// TIA Portal V18 export
FUNCTION_BLOCK "LGasp_Riordino"   // FB10300, LAD
{ S7_Optimized_Access := 'TRUE' }
VERSION : 0.1
// Da verificare:
// stored: AutoNumber true, IsIECCheckEnabled false, IsRetainMemResEnabled false, MemoryReserve 100, SetENOAutomatically false, UDAEnableTagReadback false
   VAR_INPUT
      i_lista_compilata { ExternalAccessible := 'False'; ExternalVisible := 'False'; ExternalWritable := 'False'} : Bool;   // azzerabuffer riordino e comincia a riordinare
      i_reset : Bool;
      i_svuotamentoDaPC : Bool;   // svuotamento impianto
      i_richTrasfListaPrd { ExternalAccessible := 'False'; ExternalVisible := 'False'; ExternalWritable := 'False'} : Bool;   // richiesta trasferimento lista produzione da PC
      i_mergeAbilitato { ExternalAccessible := 'False'; ExternalVisible := 'False'; ExternalWritable := 'False'} : Bool := false;   // Abilita merge quote
      I_controlloPassoLungo_ON { ExternalAccessible := 'False'; ExternalVisible := 'False'; ExternalWritable := 'False'} : Bool;   // abilita controllo passo lungo
      i_lunghezzaBanco { ExternalAccessible := 'False'; ExternalVisible := 'False'; ExternalWritable := 'False'} : LReal;
      i_quotaPrimaPunzonata { ExternalVisible := 'False'; ExternalWritable := 'False'} : LReal;
      i_correttore { ExternalVisible := 'False'; ExternalWritable := 'False'} : LReal := 1.0;
      i_passoLungoMax { ExternalVisible := 'False'; ExternalWritable := 'False'} : LReal;   // passo massimo (utilizzato per alimentatori a rulli)
   END_VAR
   VAR_OUTPUT
      o_quote_OK { ExternalAccessible := 'False'; ExternalVisible := 'False'; ExternalWritable := 'False'} : Bool;
      o_lim_max_quote { ExternalAccessible := 'False'; ExternalVisible := 'False'; ExternalWritable := 'False'} : Bool;   // raggiunto limite quote su riordino (incrementare costante "NumQuotePunzonatura" )
      o_OkTrasfListaPrd : Bool;
      o_AlmPreFineQuote : Bool;
      o_AlmFineQuote : Bool;
      o_QuotaAssoluta : "LGasp_typeBufferQuote";   // Quota assoluta
      o_QuotaAssoluta_Correttore : "LGasp_typeBufferQuote";   // Quota assoluta
      o_QuotaRelativa : "LGasp_typeBufferQuote";   // Quota relativa
      o_QuotaRelativa_Correttore : "LGasp_typeBufferQuote";   // Quota relativa con correttore
   END_VAR
   VAR_IN_OUT
      io_PunzonataEseguita { ExternalAccessible := 'False'; ExternalVisible := 'False'; ExternalWritable := 'False'} : Bool;   // cancella quota in lavoro
      io_cancella_pezzi : Bool;   // cmdbool00[8]
      io_lista_profila_nuovo_elemento : Bool;
      io_cancellazioneTotale : Bool;   // cmdbool00[11]
      io_blocca_lista_fine_prod : Bool;
      io_rich_nuovo_trasferimento : Bool;   // richiesta nuovo trasferimento all'avvio
      io_PassoInfinito : "LGasp_typeQuota";
      io_ListaProduzionePC : Array[1.."NumRigheProduzione"] of "LGasp_typeRigaProdfromPC";
      io_myprodfromPC : Array[1.."NumRigheProduzione"] of "LGasp_typeRigaProdfromPC";
      io_myprodfromPCupdate : Array[1.."NumRigheProduzione"] of DInt;
      io_myprodfromPLC : Array[1.."NumRigheProduzione"] of "LGasp_typeRigaProdfromPLC";
      io_StoricoQuotePunzonatura : Array[1.."NumQuotePunzonaturaStorico"] of "LGasp_typeBufferQuote";
      io_QuotePunzonatura : Array[1.."NumQuotePunzonatura"] of "LGasp_typeBufferQuote";
      io_StoricoRigheProdEliminate : Array[1.."NumRigheProduzione"] of "LGasp_typeRigheEliminate";
      io_pezzo_per_Lista_profila : "LGasp_typePzoListaProfila";
   END_VAR
   VAR RETAIN
      s_DM { ExternalAccessible := 'False'; ExternalVisible := 'False'; ExternalWritable := 'False'} : Struct
         OffsetPrimaPunzonata { ExternalAccessible := 'False'; ExternalVisible := 'False'; ExternalWritable := 'False'} : LReal := 0.0;   // Quota prima punzonata dopo ricompilazione
      END_STRUCT;
   END_VAR
   VAR
      s_RiordinoBufferQuote_QuickSort { ExternalAccessible := 'False'; ExternalVisible := 'False'; ExternalWritable := 'False'} : "LGasp_RiordinoBufferQuote_QuickSort";
      "s_Aggiorna&Riordina" { ExternalAccessible := 'False'; ExternalVisible := 'False'; ExternalWritable := 'False'} : Bool;   // aggiorna quote e riordina
   END_VAR
   VAR RETAIN
      s_start_riordino { ExternalAccessible := 'False'; ExternalVisible := 'False'; ExternalWritable := 'False'} : Bool;
      s_sort_riordino_OK { ExternalAccessible := 'False'; ExternalVisible := 'False'; ExternalWritable := 'False'} : Bool;
      s_lista_compilata_old { ExternalAccessible := 'False'; ExternalVisible := 'False'; ExternalWritable := 'False'} : Bool;
      s_inserire_pezzi_in_lista { ExternalAccessible := 'False'; ExternalVisible := 'False'; ExternalWritable := 'False'} : Bool;   // inserire pezzi in lista produzione
   END_VAR
   VAR
      s_firstscan_done { ExternalAccessible := 'False'; ExternalVisible := 'False'; ExternalWritable := 'False'} : Bool;
      s_ListaProduzione_ID_old { ExternalAccessible := 'False'; ExternalVisible := 'False'; ExternalWritable := 'False'} : Array[1.."NumRigheProduzione"] of DInt;
      s_index_0 { ExternalAccessible := 'False'; ExternalVisible := 'False'; ExternalWritable := 'False'} : DInt;
      s_index_1 { ExternalAccessible := 'False'; ExternalVisible := 'False'; ExternalWritable := 'False'} : DInt;
      s_index_2 { ExternalAccessible := 'False'; ExternalVisible := 'False'; ExternalWritable := 'False'} : DInt;
      s_index_3 { ExternalAccessible := 'False'; ExternalVisible := 'False'; ExternalWritable := 'False'} : DInt;
      s_index_4 { ExternalAccessible := 'False'; ExternalVisible := 'False'; ExternalWritable := 'False'} : DInt;
      s_index_5 { ExternalAccessible := 'False'; ExternalVisible := 'False'; ExternalWritable := 'False'} : DInt;
      s_index_6 { ExternalAccessible := 'False'; ExternalVisible := 'False'; ExternalWritable := 'False'} : DInt;
      s_index_7 { ExternalAccessible := 'False'; ExternalVisible := 'False'; ExternalWritable := 'False'} : DInt;
   END_VAR
   VAR RETAIN
      s_RigaProduzione_in_lavoro { ExternalAccessible := 'False'; ExternalVisible := 'False'; ExternalWritable := 'False'} : DInt;   // Indice riga di produzione in lavoro
      s_PrimaQuotaLibera { ExternalAccessible := 'False'; ExternalVisible := 'False'; ExternalWritable := 'False'} : DInt;   // Indice della prima quota NULL nella DB di riordino Quote
      s_quote_inserite { ExternalAccessible := 'False'; ExternalVisible := 'False'; ExternalWritable := 'False'} : DInt;
      s_lunghezza { ExternalAccessible := 'False'; ExternalVisible := 'False'; ExternalWritable := 'False'} : LReal;   // appoggio lunghezza pezzo i inserimento
      s_lunghezza_tot_inserita_banco { ExternalAccessible := 'False'; ExternalVisible := 'False'; ExternalWritable := 'False'} : LReal;   // lunghezza banco per inserimento pezzi
      s_tot_materiale_inserito_dopo_compilazione { ExternalAccessible := 'False'; ExternalVisible := 'False'; ExternalWritable := 'False'} : LReal;   // totale materiale inserito dopo compilazione
   END_VAR
   VAR
      s_lunghezza_banco { ExternalAccessible := 'False'; ExternalVisible := 'False'; ExternalWritable := 'False'} : LReal;
      s_QuotaNULL { ExternalAccessible := 'False'; ExternalVisible := 'False'; ExternalWritable := 'False'} : "LGasp_typeQuota";   // tipo dato NULL
      s_BufferQuotaNULL { ExternalAccessible := 'False'; ExternalVisible := 'False'; ExternalWritable := 'False'} : "LGasp_typeBufferQuote";   // tipo dato NULL
      s_RigaProduzioneNULL { ExternalAccessible := 'False'; ExternalVisible := 'False'; ExternalWritable := 'False'} : "LGasp_typeRigaProdfromPC";   // tipo dato NULL
      s_mem_trasf_lista_da_PC { ExternalAccessible := 'False'; ExternalVisible := 'False'; ExternalWritable := 'False'} : Bool;
   END_VAR
   VAR RETAIN
      s_ID_righe_produzione { ExternalAccessible := 'False'; ExternalVisible := 'False'; ExternalWritable := 'False'} : Array[1.."NumRigheProduzione"] of DInt;
      s_quotaTestaInserita { ExternalAccessible := 'False'; ExternalVisible := 'False'; ExternalWritable := 'False'} : Bool;
      s_mem_quota { ExternalAccessible := 'False'; ExternalVisible := 'False'; ExternalWritable := 'False'} : LReal;
      s_appQuota { ExternalAccessible := 'False'; ExternalVisible := 'False'; ExternalWritable := 'False'} : LReal;
      s_count { ExternalAccessible := 'False'; ExternalVisible := 'False'; ExternalWritable := 'False'} : DInt;
      s_num_pzi_banco { ExternalAccessible := 'False'; ExternalVisible := 'False'; ExternalWritable := 'False'} : Int;
   END_VAR
   VAR
      s_FPPreFine { ExternalAccessible := 'False'; ExternalVisible := 'False'; ExternalWritable := 'False'} : Bool;
      s_ResetPassoInfinito { ExternalAccessible := 'False'; ExternalVisible := 'False'; ExternalWritable := 'False'} : Bool;
      s_primoTrasferimentoEseguito { ExternalAccessible := 'False'; ExternalVisible := 'False'; ExternalWritable := 'False'} : Bool;
      s_passoLungoON : Bool;
   END_VAR
   VAR_TEMP
      t_passoLungoMax : LReal;
   END_VAR
   VAR_TEMP   // added for the SCL form of the ladder/FBD networks
      _w1 : Bool;
   END_VAR
BEGIN

REGION Network 1 (SCL): Descrizione
   //================================================================================
   // Gasparini Spa
   //--------------------------------------------------------------------------------
   // Libreria: LGaspQset_Riordino
   // Funzionalità: Funzione globale per gestione riordino quote
   // Commessa in cui è stata testata: YYXXNNNNN
   // Programmatore di riferimento per test: XXXXXX
   //--------------------------------------------------------------------------------
   // Change log table:
   // Versione Data        Autore          Modifiche
   // 01.00.03 02.07.2020  P.Toaldo        Aggiornamento dopo test quote con PC
   // 01.00.04 22/03/2021  Lcg             Banco di punzonatura per calcoli quote deve essere il doppio di quello reale
   // 01.00.05 08/04/2021  Lcg             Inserito un pulsante da PC che esegue la cancellazione totale
   // 01.00.06 27/05/2021  P.Toaldo        Correzione aggiornamento quota dopo set "io_PunzonataEseguita". Micron 305
   // 01.00.06 27/05/2021  Lcg             Correzione uscita "Sort" blocco riordino che non era ritentiva  Micron 305
   // 01.00.07 03/06/2021  Lcg             Correzione errore prefine lista e aggiunto blocco lista di produzione a fine pezzi
   // 01.00.08 10/06/2021  Lcg             Reset passo infinito con cancellazione lista
   // 01.00.09 28/06/2021  Lcg             Corretto errore cancellazione passo infinito con nuova compilazione
   // 01.00.10 06/07/2021  Lcg             Corretto errore nuovo trasferimento all'avvio del PC seg 18
   // 01.00.11 28/01/2022  Lcg             Aggiunto il reset dell'area di memoria passo infinito con primo trasferimento e lista non compilata
   // 01.00.12 02/03/2022  Lcg/A.Donà      Aggiunto il numero del pezzo a cui fa riferimento la quota. In state aggiunto se la quota è una quota di sincronismo.
   //                                      Aggiunto nome articolo nella struttura per passaggio a lista profila e ad eventuale tracking (210100012)
   // 01.00.13 10/10/2022  Lcg             Passaggio nuovi dati option.DINT, options.Lreal, options.Str in lista profila
   // 01.00.14 24/01/2023  Lcg             Aggiunto "i_quotaPrimaPunzonata" alla prima quota se era un passo infinito perchè non veniva sommata
   // 01.00.15 14/03/2023  Lcg             Corretto errore che all'avvio azzerava i pezzi fatti dopo uno snapshot di L1_prd (22010003)
   // 01.00.16 17/03/2023  Lcg             Eliminata la funzionalità lunghezza pezzi non multipla del passo alimentatore usata solo su Micron 303 perchè creava confusione con lenght e nominal lenght 
   //                                      in quanto lenght comprende lo sfrido e nominal lenght è senza sfrido. Questo causava un errore nella visualizzazione del numero pezzo della lista profila.
   //                                      Corretto errore "Allarme fine pezzi" all'accensione, si attende il primo trasferimento. 
   // 01.00.17 20/04/2023  Lcg             Aggiunta gestione passo lungo, si può abilitare una funzione che in caso di quota maggiore di i_passoLungoMax la quota viene ridotta
   //                                      in sottopassi di grandezza massima i_passoLungoMax (SIPPA 220100034). Passo lungo e passo infinito non possono coesistere.
   // 01.00.18 09/05/2023  Lcg             Modificato blocco inserimento righe PC dopo preavviso fine lista perchè se veniva premuto reset prima di inserire la riga non era più possibile
   //                                      eseguire l'inserimento (dierre 210100104)
   // 
   //-------------------------------------------------------------------------------
   //================================================================================
END_REGION

REGION Network 2 (SCL): Lunghezza banco di punzonatura + quota primapunzonata
   // la lunghezza del banco di punzonatura sul nuovo riordino quote deve essere uguale alla lunghezza reale del banco per 2 altrimenti possono capitare casi per cui l'inserimento delle nuove quote è tardivo
   //lunghezza banco
   #s_lunghezza_banco := #i_lunghezzaBanco * 2.0;

   //quota prima punz
   #s_DM.OffsetPrimaPunzonata := #i_quotaPrimaPunzonata;

   //valore quota/passo massimo
   #t_passoLungoMax := #i_passoLungoMax;
END_REGION

REGION Network 3 (SCL): Appoggio Produzione dal PC sulla produzione del PLC


   IF #i_richTrasfListaPrd THEN
       #s_mem_trasf_lista_da_PC := TRUE;
   END_IF;

   IF NOT #i_richTrasfListaPrd AND #s_mem_trasf_lista_da_PC THEN
       #s_mem_trasf_lista_da_PC := FALSE;
       #io_myprodfromPC :=  #io_ListaProduzionePC;
   END_IF;
END_REGION

REGION Network 4 (SCL): Su fronte compilazione lista -> cancello tutto il DB riordino quote e lancio riordino
   IF #i_lista_compilata AND (NOT #s_lista_compilata_old) AND NOT #i_richTrasfListaPrd THEN

       FOR #s_index_1 := 1 TO "NumQuotePunzonatura" DO // Statement section IF
           #io_QuotePunzonatura[#s_index_1] := #s_BufferQuotaNULL;
       END_FOR;

       // cancella storico
       FOR #s_index_1 := 1 TO "NumQuotePunzonaturaStorico" DO // Statement section IF
           #io_StoricoQuotePunzonatura[#s_index_1] := #s_BufferQuotaNULL;
       END_FOR;

       // Aggiorno il numero di pezzi inseriti nel riordino quote = pezzi fatti
       FOR #s_index_1 := 1 TO "NumRigheProduzione" DO
           #io_myprodfromPLC[#s_index_1].pzinseritinelriordinoquote := #io_myprodfromPLC[#s_index_1].pzfatti;
       END_FOR;
       #s_tot_materiale_inserito_dopo_compilazione := #s_DM.OffsetPrimaPunzonata;
       #s_lunghezza_tot_inserita_banco := 0.0;
       #s_quotaTestaInserita := False;
       #s_passoLungoON := false;
       #s_num_pzi_banco := 0;

       #"s_Aggiorna&Riordina" := true;
   END_IF;

   IF #i_lista_compilata = false AND #s_lista_compilata_old = true THEN

       FOR #s_index_1 := 1 TO "NumQuotePunzonatura" DO // Statement section IF
           #io_QuotePunzonatura[#s_index_1] := #s_BufferQuotaNULL;
       END_FOR;

       // Aggiorno il numero di pezzi inseriti nel riordino quote = pezzi fatti
       FOR #s_index_1 := 1 TO "NumRigheProduzione" DO
           #io_myprodfromPLC[#s_index_1].pzinseritinelriordinoquote := #io_myprodfromPLC[#s_index_1].pzfatti;
       END_FOR;

       #s_tot_materiale_inserito_dopo_compilazione := #s_DM.OffsetPrimaPunzonata;
       #s_lunghezza_tot_inserita_banco := 0.0;
       #s_quotaTestaInserita := False;
       #s_passoLungoON := false;
       #s_num_pzi_banco := 0;

   END_IF;

   #s_lista_compilata_old := #i_lista_compilata;
END_REGION

REGION Network 5 (SCL): Cancellazione totale da pulsante in pagina di produzione che esegue la cancellazione totale
       IF #io_cancellazioneTotale THEN

           //cancella quote punzonatura
           FOR #s_index_1 := 1 TO "NumQuotePunzonatura" DO // Statement section IF
               #io_QuotePunzonatura[#s_index_1] := #s_BufferQuotaNULL;
           END_FOR;

           //cancello tutto
           FOR #s_index_1 := 1 TO "NumRigheProduzione" DO
               #io_myprodfromPLC[#s_index_1].pzinseritinelriordinoquote := 0;
               #io_myprodfromPLC[#s_index_1].pzfatti := 0;

               #io_myprodfromPC[#s_index_1].ID := 0;
               #io_myprodfromPC[#s_index_1].piecestodo := 0;
               #io_myprodfromPC[#s_index_1].tipoarticolo := 0;

           END_FOR;

           #io_cancellazioneTotale := false;

       END_IF;
END_REGION

REGION Network 6 (SCL): Cancellazione aree passo infinito con primo trasferimento e lista non compilata in quanto il PC non le cancella
           //Nessun trasferimento in corso
           IF NOT #i_richTrasfListaPrd THEN
               #s_ResetPassoInfinito := false;
           END_IF;

           //con fronte trasferimento e lista non compilata azzero l'area del passo infinito
           IF NOT #i_lista_compilata AND #i_richTrasfListaPrd AND NOT #s_ResetPassoInfinito THEN

               #s_ResetPassoInfinito := true;

               //reset passo infinito 
               #io_PassoInfinito.quotax := -1;
               #io_PassoInfinito.quotay := -1;

               //reset dei punzoni del passo infinito
               FOR #s_index_1 := 1 TO 16 DO
                   #io_PassoInfinito.mouldea[#s_index_1] := false;
                   #io_PassoInfinito.mouldeb[#s_index_1] := false;
                   #io_PassoInfinito.mouldec[#s_index_1] := false;
                   #io_PassoInfinito.moulded[#s_index_1] := false;
               END_FOR;

               #io_PassoInfinito.infinitystep := false;

           END_IF;
END_REGION

REGION Network 7 (SCL): Riga di produzione in lavoro
   FOR #s_index_1 := 1 TO "NumRigheProduzione" DO
       IF #io_myprodfromPLC[#s_index_1].pzfatti < #io_myprodfromPC[#s_index_1].piecestodo THEN
           #s_RigaProduzione_in_lavoro := #s_index_1;
           EXIT;
       END_IF;
   END_FOR;
END_REGION

REGION Network 8 (SCL): Prima quota libera nel DB di riordino quote
   FOR #s_index_1 := 1 TO "NumQuotePunzonatura" DO
       IF NOT(#io_QuotePunzonatura[#s_index_1].quota.state.quotavalida) THEN
           #s_PrimaQuotaLibera := #s_index_1;
           EXIT;
       END_IF;
   END_FOR;
END_REGION

REGION Network 9: Reset allarme limite massimo quote inserite con togli compilazione
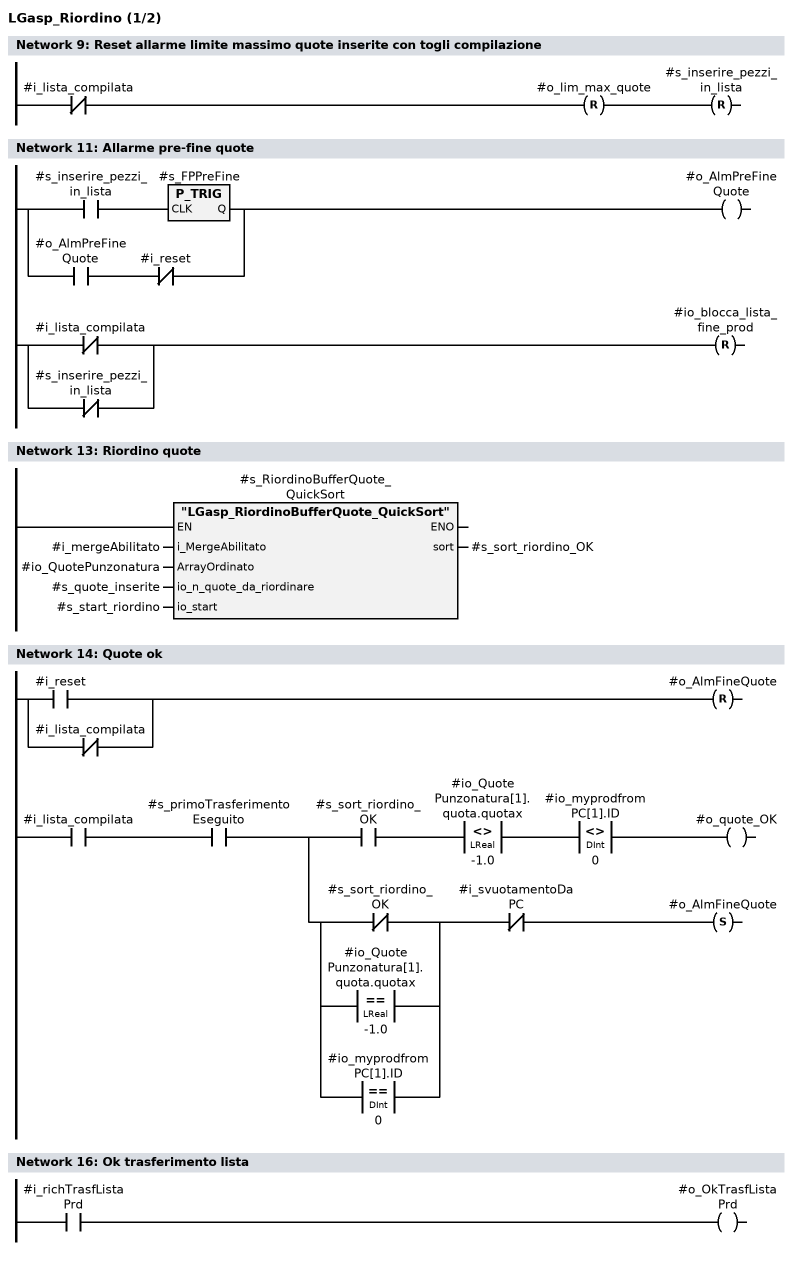
   RUNG wire#powerrail
      I_Contact( #i_lista_compilata )
      R_Coil( #o_lim_max_quote )
      R_Coil( #s_inserire_pezzi_in_lista )
   END_RUNG
   // the same network as SCL:
   IF NOT #i_lista_compilata THEN
       #o_lim_max_quote := FALSE;
       #s_inserire_pezzi_in_lista := FALSE;
   END_IF;
END_REGION

REGION Network 10 (SCL): Lista quote con le quote con articoli fino a riempire la lunghezza del banco di punzonatura
   // rilancio controllo per verifica pre-fine quote
   IF #i_reset AND #o_AlmPreFineQuote THEN
       #"s_Aggiorna&Riordina" := TRUE;
   END_IF;


   IF #"s_Aggiorna&Riordina" AND #s_primoTrasferimentoEseguito THEN
       #io_PunzonataEseguita := false;
       #s_inserire_pezzi_in_lista := false;
       #s_quote_inserite := #s_PrimaQuotaLibera - 1;



       // Se presente passo infinito inserisco la prima quota
       IF #s_quote_inserite = 0 AND #io_PassoInfinito.infinitystep THEN

           // INSERISCO QUOTA SU RIORDINO
           #s_quote_inserite := #s_quote_inserite + 1;
           #io_QuotePunzonatura[#s_quote_inserite].quota := #io_PassoInfinito;
           //24.01.2023 lcg
           //aggiungo prima quota al primo passo infinito
           #io_QuotePunzonatura[#s_quote_inserite].quota.quotax := #io_QuotePunzonatura[#s_quote_inserite].quota.quotax + #i_quotaPrimaPunzonata;

       END_IF;

       //verifico se la prima quota supera il passo massimo 
       IF #s_quote_inserite = 0 AND #I_controlloPassoLungo_ON AND NOT #io_PassoInfinito.infinitystep AND NOT #s_passoLungoON THEN

           #s_appQuota := #io_myprodfromPC[1].article.prepunchingquota[1].quotax + #i_quotaPrimaPunzonata;

           IF #s_appQuota > #i_passoLungoMax THEN

               // INSERISCO QUOTA SU RIORDINO

               #s_quote_inserite := #s_quote_inserite + 1;
               //cancello tutti i cassetti
               #io_QuotePunzonatura[1].quota := #s_QuotaNULL;
               #io_QuotePunzonatura[#s_quote_inserite].quota.quotax := #i_passoLungoMax;
               #s_passoLungoON := true;

           END_IF;
       END_IF;

       // Inserisco le quote degli articoli fino al riempimento del banco di punzonatura
       FOR #s_index_1 := 1 TO "NumRigheProduzione" DO
           IF #io_myprodfromPLC[#s_index_1].pzinseritinelriordinoquote < #io_myprodfromPC[#s_index_1].piecestodo THEN
               FOR #s_index_2 := #io_myprodfromPLC[#s_index_1].pzinseritinelriordinoquote + 1 TO #io_myprodfromPC[#s_index_1].piecestodo DO
                   IF #s_lunghezza_tot_inserita_banco < #s_lunghezza_banco OR #s_num_pzi_banco < 2 THEN
                       // Inserisco tutte le punzonate dell'articolo in riga di produzione
                       FOR #s_index_3 := 1 TO "NumPunzonateArticolo" DO

                           // Controllo che la quota dell'articolo sia valida
                           IF #io_myprodfromPC[#s_index_1].article.prepunchingquota[#s_index_3].state.quotavalida AND NOT (#o_lim_max_quote)  THEN

                               //24.01.2023 Lcg: Tolta l'istruzione che non metteva nel riordino le quote di testa dopo la prima (Dierre 104)
                               //IF (NOT #s_quotaTestaInserita OR NOT #io_myprodfromPC[#s_index_1].article.prepunchingquota[#s_index_3].state.quotatagliotesta) THEN

                                   IF #io_myprodfromPC[#s_index_1].article.prepunchingquota[#s_index_3].state.quotatagliotesta THEN
                                       #s_quotaTestaInserita := TRUE;
                                   END_IF;

                                   // incrementa quote inserite
                                   #s_quote_inserite := #s_quote_inserite + 1;

                                   // Aggiorno articolo, general , quota e testo stampa

                                   #io_QuotePunzonatura[#s_quote_inserite].general := #io_myprodfromPC[#s_index_1].article.general;
                                   #io_QuotePunzonatura[#s_quote_inserite].quota := #io_myprodfromPC[#s_index_1].article.prepunchingquota[#s_index_3];
                                   #io_QuotePunzonatura[#s_quote_inserite].general.print := #io_myprodfromPC[#s_index_1].article.general.print;
                                   #io_QuotePunzonatura[#s_quote_inserite].ID := #io_myprodfromPC[#s_index_1].ID;
                                   //numero del pezzo a cui fa riferimento la quota
                                   #io_QuotePunzonatura[#s_quote_inserite].n_piece := #s_index_2;

                                   // alla quota X aggiungo l'offset di partenza
                                   #io_QuotePunzonatura[#s_quote_inserite].quota.quotax := (#io_QuotePunzonatura[#s_quote_inserite].quota.quotax) + #s_tot_materiale_inserito_dopo_compilazione;



                                   // memorizzo lunghezza pezzo dell'ultima quota
                                   IF #io_QuotePunzonatura[#s_quote_inserite].quota.state.ultimaquotapezzo THEN
                                       #s_lunghezza := #io_QuotePunzonatura[#s_quote_inserite].general.lenght;
                                       EXIT;
                                   END_IF;

                                   // verifica limite quote nel riordino raggiunte
                                   IF #s_quote_inserite >= "NumQuotePunzonatura" THEN
                                       #o_lim_max_quote := TRUE;
                                   END_IF;
                               //END_IF;
                           ELSE
                               EXIT;
                           END_IF;
                       END_FOR;

                       // Aggiungo un pezzo ai pezzi presi in carico dal riordino quote per la riga di produzione in lavoro
                       #io_myprodfromPLC[#s_index_1].pzinseritinelriordinoquote := #io_myprodfromPLC[#s_index_1].pzinseritinelriordinoquote + 1;

                       // aggiorno totale materiale inserito in banco di punzonatura
                       #s_lunghezza_tot_inserita_banco := #s_lunghezza_tot_inserita_banco + #s_lunghezza ;
                       #s_num_pzi_banco := #s_num_pzi_banco+1;

                       // aggiorno totale materiale inserito da dopo compilazione
                       #s_tot_materiale_inserito_dopo_compilazione := #s_tot_materiale_inserito_dopo_compilazione + #s_lunghezza;

                   END_IF;
               END_FOR;
           END_IF;
       END_FOR;

       // verifica fine pezzi
       IF #s_lunghezza_tot_inserita_banco < #s_lunghezza_banco OR #s_num_pzi_banco<2 THEN
           #s_inserire_pezzi_in_lista := true;
       END_IF;



       // comando riordino quote
       #"s_Aggiorna&Riordina" := FALSE;
       #s_start_riordino := true;
   END_IF;
END_REGION

REGION Network 11: Allarme pre-fine quote
   RUNG wire#powerrail
      Contact( #s_inserire_pezzi_in_lista )
      P_Trig( #s_FPPreFine )
      wire#w1
      Coil( #o_AlmPreFineQuote )
   END_RUNG
   RUNG wire#powerrail
      Contact( #o_AlmPreFineQuote )
      I_Contact( #i_reset )
   END_RUNG wire#w1
   RUNG wire#powerrail
      I_Contact( #i_lista_compilata )
      wire#w2
      R_Coil( #io_blocca_lista_fine_prod )
   END_RUNG
   RUNG wire#powerrail
      I_Contact( #s_inserire_pezzi_in_lista )
   END_RUNG wire#w2
   // the same network as SCL:
   #_w1 := #s_inserire_pezzi_in_lista AND NOT #s_FPPreFine;   // rising edge
   #s_FPPreFine := #s_inserire_pezzi_in_lista;
   #o_AlmPreFineQuote := #_w1 OR (#o_AlmPreFineQuote AND NOT #i_reset);
   IF NOT #i_lista_compilata OR NOT #s_inserire_pezzi_in_lista THEN
       #io_blocca_lista_fine_prod := FALSE;
   END_IF;
END_REGION

REGION Network 12 (SCL): Quota eseguita + inserimento nuova quota + riordino
   // comando quota eseguita ->
   // 1 - popolare il DB StoricoQuotePunzonatura con la quota appena cancellata
   // 2 - verificare se è l'ultima quota del pezzo
   // 3 - cancellare prima quota della lista punzonatura

   IF #io_PunzonataEseguita THEN
       #s_count := #s_count + 1;

       // ****************************************
       // aggiornamento DB StoricoQuotePunzonatura 
       // ****************************************

       // Shifto array di un posto per liberare il primo record dell'array
       // NB: record [1] è il più recente
       FOR #s_index_1 := "NumQuotePunzonaturaStorico" TO 2 BY -1 DO
           #io_StoricoQuotePunzonatura[#s_index_1] := #io_StoricoQuotePunzonatura[#s_index_1 - 1];
       END_FOR;

       // Scrivo il primo record dell'array = quota da cancellare
       #io_StoricoQuotePunzonatura[1] := #io_QuotePunzonatura[1];

       // verifico se è l'ultima quota del pezzo
       IF #io_QuotePunzonatura[1].quota.state.ultimaquotapezzo THEN

           // aggiona dati per lista profila
           #io_pezzo_per_Lista_profila.ID := #io_QuotePunzonatura[1].ID;

           //gestione lista profila con articolo a passo e non a passo
           //articolo a passo dello stampo
           //modalità usata in micron 303 dove la lunghezza del pezzo era diversa dal passo fisso dell'alimentatore
           //IF (#io_QuotePunzonatura[1].general.lenght = #io_QuotePunzonatura[1].general.nominal_lenght) OR #io_QuotePunzonatura[1].general.nominal_lenght = -1.0 THEN
           //    #io_pezzo_per_Lista_profila.lenght := #io_QuotePunzonatura[1].general.lenght;
           #io_pezzo_per_Lista_profila.NumeroPezzo := #io_myprodfromPLC[1].pzfatti + 1;
           //ELSE
           //articolo non a passo dello stampo
           #io_pezzo_per_Lista_profila.lenght := #io_QuotePunzonatura[1].general.nominal_lenght;
           //   #io_pezzo_per_Lista_profila.NumeroPezzo := #io_myprodfromPLC[1].pzfattinopasso + 1;
           //END_IF;

           #io_pezzo_per_Lista_profila.cutoffset := #io_QuotePunzonatura[1].general.cutoffset;
           #io_pezzo_per_Lista_profila.options := #io_QuotePunzonatura[1].general.options;
           #io_pezzo_per_Lista_profila.options_dint := #io_myprodfromPC[#s_RigaProduzione_in_lavoro].article.general.options_dint;
           #io_pezzo_per_Lista_profila.options_lreal := #io_myprodfromPC[#s_RigaProduzione_in_lavoro].article.general.options_lreal;
           #io_pezzo_per_Lista_profila.options_str := #io_myprodfromPC[#s_RigaProduzione_in_lavoro].article.general.options_str;
           #io_lista_profila_nuovo_elemento := true;

           // incremento pezzi fatti
           #io_myprodfromPLC[#s_RigaProduzione_in_lavoro].pzfatti := #io_myprodfromPLC[#s_RigaProduzione_in_lavoro].pzfatti + 1;
           // aggiorna lunghezza totale inserita su banco punzonatura
           #s_lunghezza_tot_inserita_banco := #s_lunghezza_tot_inserita_banco - #io_QuotePunzonatura[1].general.lenght;
           #s_num_pzi_banco := #s_num_pzi_banco - 1;
       END_IF;

       // se quota passo infinito riaggiungo la quota altrimenti la elimino
       IF NOT #I_controlloPassoLungo_ON THEN

           // se quota passo infinito riaggiungo la quota altrimenti la elimino
           IF #io_QuotePunzonatura[1].quota.infinitystep THEN

               #s_mem_quota := #io_QuotePunzonatura[1].quota.quotax;
               #io_QuotePunzonatura[1].quota := #io_PassoInfinito;
               #io_QuotePunzonatura[1].quota.quotax := #s_mem_quota + #io_PassoInfinito.quotax;

           ELSE
               FOR #s_index_6 := 1 TO "NumQuotePunzonatura" - 1 DO
                   #io_QuotePunzonatura[#s_index_6] := #io_QuotePunzonatura[#s_index_6 + 1];
               END_FOR;
               #io_QuotePunzonatura[NumQuotePunzonatura] := #s_BufferQuotaNULL;
           END_IF;

       ELSE

           //entro qui se ho il controllo passo lungo
           IF ((#io_QuotePunzonatura[2].quota.quotax - #io_QuotePunzonatura[1].quota.quotax) > #i_passoLungoMax) AND #io_QuotePunzonatura[2].quota.quotax > 0.0 THEN

               //appoggio quota
               #s_mem_quota := #io_QuotePunzonatura[1].quota.quotax;
               //cancello tutti i cassetti
               #io_QuotePunzonatura[1].quota := #s_QuotaNULL;
               #io_QuotePunzonatura[1].quota.quotax := #s_mem_quota + #i_passoLungoMax;

           ELSE
               FOR #s_index_6 := 1 TO "NumQuotePunzonatura" - 1 DO
                   #io_QuotePunzonatura[#s_index_6] := #io_QuotePunzonatura[#s_index_6 + 1];
               END_FOR;
               #io_QuotePunzonatura[NumQuotePunzonatura] := #s_BufferQuotaNULL;
           END_IF;

       END_IF;

       // comando aggiornamento quote + riordino
       #"s_Aggiorna&Riordina" := true;

       //blocco inserimento righe dopo ripartenza e prefine quote attivo
       IF #s_inserire_pezzi_in_lista AND NOT #o_AlmPreFineQuote THEN
           #io_blocca_lista_fine_prod := true;
       END_IF;

   END_IF;
END_REGION

REGION Network 13: Riordino quote
   RUNG wire#powerrail
      #s_RiordinoBufferQuote_QuickSort(i_MergeAbilitato := #i_mergeAbilitato, ArrayOrdinato := #io_QuotePunzonatura, io_n_quote_da_riordinare := #s_quote_inserite, io_start := #s_start_riordino, sort => #s_sort_riordino_OK)
   END_RUNG
   // the same network as SCL:
   #s_RiordinoBufferQuote_QuickSort(i_MergeAbilitato := #i_mergeAbilitato,   // "LGasp_RiordinoBufferQuote_QuickSort"
                           ArrayOrdinato := #io_QuotePunzonatura,
                           io_n_quote_da_riordinare := #s_quote_inserite,
                           io_start := #s_start_riordino,
                           sort => #s_sort_riordino_OK);
END_REGION

REGION Network 14: Quote ok
   RUNG wire#powerrail
      Contact( #i_reset )
      wire#w1
      R_Coil( #o_AlmFineQuote )
   END_RUNG
   RUNG wire#powerrail
      I_Contact( #i_lista_compilata )
   END_RUNG wire#w1
   RUNG wire#powerrail
      Contact( #i_lista_compilata )
      Contact( #s_primoTrasferimentoEseguito )
      wire#w2
      Contact( #s_sort_riordino_OK )
      { S7_Templates := "SrcType := LReal" } NE_Contact(in1 := #io_QuotePunzonatura[1].quota.quotax, in2 := -1.0)
      { S7_Templates := "SrcType := DInt" } NE_Contact(in1 := #io_myprodfromPC[1].ID, in2 := 0)
      Coil( #o_quote_OK )
   END_RUNG
   RUNG wire#w2
      I_Contact( #s_sort_riordino_OK )
      wire#w3
      I_Contact( #i_svuotamentoDaPC )
      S_Coil( #o_AlmFineQuote )
   END_RUNG
   RUNG wire#w2
      { S7_Templates := "SrcType := LReal" } EQ_Contact(in1 := #io_QuotePunzonatura[1].quota.quotax, in2 := -1.0)
   END_RUNG wire#w3
   RUNG wire#w2
      { S7_Templates := "SrcType := DInt" } EQ_Contact(in1 := #io_myprodfromPC[1].ID, in2 := 0)
   END_RUNG wire#w3
   // the same network as SCL:
   IF #i_reset OR NOT #i_lista_compilata THEN #o_AlmFineQuote := FALSE; END_IF;
   #_w1 := #i_lista_compilata AND #s_primoTrasferimentoEseguito;
   #o_quote_OK := #_w1 AND #s_sort_riordino_OK AND (#io_QuotePunzonatura[1].quota.quotax <> (-1.0)) AND (#io_myprodfromPC[1].ID <> 0);
   IF #_w1 AND (NOT #s_sort_riordino_OK OR (#io_QuotePunzonatura[1].quota.quotax = (-1.0)) OR (#io_myprodfromPC[1].ID = 0)) AND NOT #i_svuotamentoDaPC THEN
       #o_AlmFineQuote := TRUE;
   END_IF;
END_REGION

REGION Network 15 (SCL): Elimina righe terminate (attenzione le elimino solo da parte PLC )
   IF NOT #s_mem_trasf_lista_da_PC AND #s_primoTrasferimentoEseguito THEN

       IF (#io_myprodfromPLC[1].pzfatti >= #io_myprodfromPC[1].piecestodo) AND (#io_myprodfromPC[1].piecestodo > 0) THEN


           //salvataggio ID e pezzi fatti della riga appena completata: serve al PC per impostare correttamente i pezzi fatti
           //nelle righe eliminate
           //spostamento delle righe 
           FOR #s_index_5 := 0 TO "NumRigheProduzione" - 2 DO
               #io_StoricoRigheProdEliminate[NumRigheProduzione - #s_index_5] := #io_StoricoRigheProdEliminate[NumRigheProduzione - #s_index_5 - 1];
           END_FOR;

           //salvataggio ID e pezzi fatti prima di eliminare la riga di produzione
           #io_StoricoRigheProdEliminate[1].ID := #io_myprodfromPC[1].ID;
           #io_StoricoRigheProdEliminate[1].pzfatti := #io_myprodfromPLC[1].pzfatti;

           //cancella pezzi fatti
           #io_myprodfromPLC[1].pzfatti := 0;

           //salvataggio nuovi dati

           //sposta le righe di produzione
           FOR #s_index_5 := 1 TO "NumRigheProduzione" - 1 DO
               #io_myprodfromPC[#s_index_5] := #io_myprodfromPC[#s_index_5 + 1];
               #io_myprodfromPLC[#s_index_5] := #io_myprodfromPLC[#s_index_5 + 1];
           END_FOR;

           #io_myprodfromPC[NumRigheProduzione] := #s_RigaProduzioneNULL;

       END_IF;
   END_IF;
END_REGION

REGION Network 16: Ok trasferimento lista
   RUNG wire#powerrail
      Contact( #i_richTrasfListaPrd )
      Coil( #o_OkTrasfListaPrd )
   END_RUNG
   // the same network as SCL:
   #o_OkTrasfListaPrd := #i_richTrasfListaPrd;
END_REGION

REGION Network 17 (SCL): Cancella pezzi fatti
   IF NOT #i_lista_compilata AND #io_cancella_pezzi THEN
       FOR #s_index_7 := 1 TO "NumRigheProduzione" DO
           #io_myprodfromPLC[#s_index_7].pzfatti := 0;
           #io_myprodfromPLC[#s_index_7].pzinseritinelriordinoquote := 0;
       END_FOR;
   END_IF;

   #io_cancella_pezzi := false;
END_REGION

REGION Network 18 (SCL): Aggiornamento pezzi da fare durante la marcia
   // Controllo se sono stati modificati i pezzi da fare in pagina di produzione e aggiorno le righe di produzione con i nuovi pezzi
       FOR #s_index_7 := 1 TO "NumRigheProduzione" DO

           IF #io_myprodfromPCupdate[#s_index_7] > 0 AND #io_myprodfromPCupdate[#s_index_7] > #io_myprodfromPLC[#s_index_7].pzinseritinelriordinoquote THEN
               #io_myprodfromPC[#s_index_7].piecestodo := #io_myprodfromPCupdate[#s_index_7];
           END_IF;
           #io_myprodfromPCupdate[#s_index_7] := 0;

       END_FOR;
END_REGION

REGION Network 19 (SCL): Memoria ID prima riga per riallineamento all'accensione
   IF NOT #s_firstscan_done THEN

       FOR #s_index_0 := 1 TO "NumRigheProduzione" DO
           #io_myprodfromPC[#s_index_0].ID := #s_ID_righe_produzione[#s_index_0];
       END_FOR;

       #io_rich_nuovo_trasferimento := true;
       #s_firstscan_done := true;

   END_IF;

   IF #s_firstscan_done AND NOT #io_rich_nuovo_trasferimento THEN
       FOR #s_index_0 := 1 TO "NumRigheProduzione" DO
           #s_ID_righe_produzione[#s_index_0] := #io_myprodfromPC[#s_index_0].ID;
       END_FOR;
       #s_primoTrasferimentoEseguito := true;
   END_IF;
END_REGION

REGION Network 20: Quote prossima lavorazione
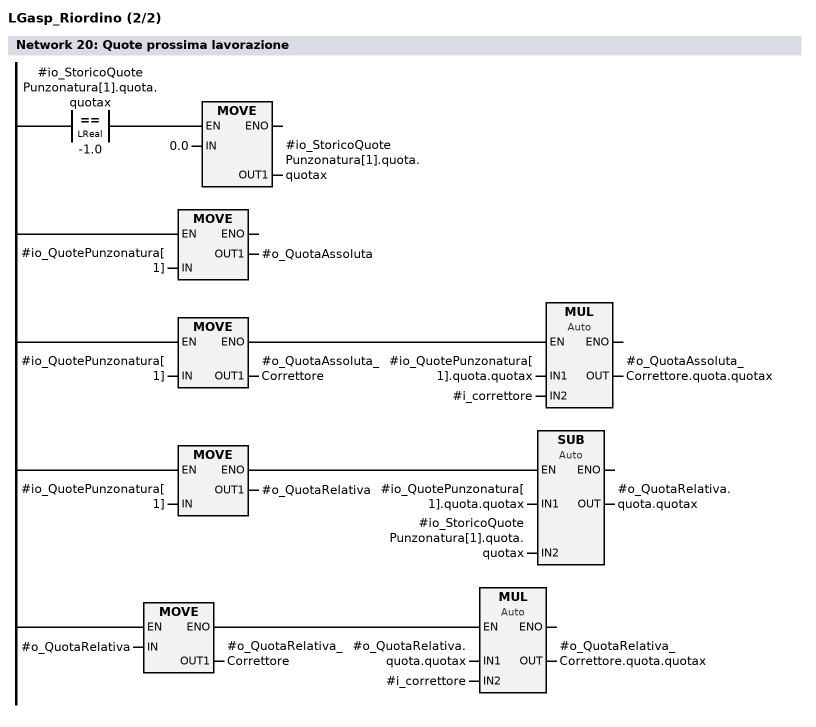
   RUNG wire#powerrail
      { S7_Templates := "SrcType := LReal" } EQ_Contact(in1 := #io_StoricoQuotePunzonatura[1].quota.quotax, in2 := -1.0)
      Move(in := 0.0, out1 => #io_StoricoQuotePunzonatura[1].quota.quotax)
   END_RUNG
   RUNG wire#powerrail
      Move(in := #io_QuotePunzonatura[1], out1 => #o_QuotaAssoluta)
   END_RUNG
   RUNG wire#powerrail
      Move(in := #io_QuotePunzonatura[1], out1 => #o_QuotaAssoluta_Correttore)
      Mul(in1 := #io_QuotePunzonatura[1].quota.quotax, in2 := #i_correttore, out => #o_QuotaAssoluta_Correttore.quota.quotax)
   END_RUNG
   RUNG wire#powerrail
      Move(in := #io_QuotePunzonatura[1], out1 => #o_QuotaRelativa)
      Sub(in1 := #io_QuotePunzonatura[1].quota.quotax, in2 := #io_StoricoQuotePunzonatura[1].quota.quotax, out => #o_QuotaRelativa.quota.quotax)
   END_RUNG
   RUNG wire#powerrail
      Move(in := #o_QuotaRelativa, out1 => #o_QuotaRelativa_Correttore)
      Mul(in1 := #o_QuotaRelativa.quota.quotax, in2 := #i_correttore, out => #o_QuotaRelativa_Correttore.quota.quotax)
   END_RUNG
   // the same network as SCL:
   IF #io_StoricoQuotePunzonatura[1].quota.quotax = (-1.0) THEN
       #io_StoricoQuotePunzonatura[1].quota.quotax := 0.0;
   END_IF;
   #o_QuotaAssoluta := #io_QuotePunzonatura[1];
   #o_QuotaAssoluta_Correttore := #io_QuotePunzonatura[1];
   #o_QuotaAssoluta_Correttore.quota.quotax := #io_QuotePunzonatura[1].quota.quotax * #i_correttore;
   #o_QuotaRelativa := #io_QuotePunzonatura[1];
   #o_QuotaRelativa.quota.quotax := #io_QuotePunzonatura[1].quota.quotax - #io_StoricoQuotePunzonatura[1].quota.quotax;
   #o_QuotaRelativa_Correttore := #o_QuotaRelativa;
   #o_QuotaRelativa_Correttore.quota.quotax := #o_QuotaRelativa.quota.quotax * #i_correttore;
END_REGION
END_FUNCTION_BLOCK
